TYPE "CLEANING HOPPER"
// stored: IsFailsafeCompliant false
   STRUCT
      FAULTED : Bool;
      "START GENERAL CONDITIONS" : Bool;
      "START GENERAL CONDITIONS HELP" : Bool;
      "START INITIAL CONDITIONS" : Bool;
      "START INITIAL CONDITIONS HELP" : Bool;
      "START MANUAL REQUEST" : Bool;
      "FEEDBACK ON" : Bool;
      "START SEMI REQUEST" : Bool;
      "START AUTO REQUEST" : Bool;
      "START GLOBAL REQUEST" : Bool;
      "START COMMAND" : Bool;
      "SYSTEM ON" : Bool;
      "STOP GENERAL CONDITIONS" : Bool;
      "STOP GENERAL CONDITIONS HELP" : Bool;
      "STOP INITIAL CONDITIONS" : Bool;
      "STOP INITIAL CONDITIONS HELP" : Bool;
      "STOP MANUAL REQUEST" : Bool;
      "STOP SEMI REQUEST" : Bool;
      "STOP AUTO REQUEST" : Bool;
      "STOP GLOBAL REQUEST" : Bool;
      "STOP COMMAND" : Bool;
      STOPPED : Bool;
      "FEEDBACK OFF" : Bool;
   END_STRUCT;
END_TYPE

TYPE "FEED HOPPER"
// stored: IsFailsafeCompliant false
   STRUCT
      FAULTED : Bool;   // Faulted
      "START GENERAL CONDITIONS" : Bool;   // Start General Conditions
      "START GENERAL CONDITIONS HELP" : Bool;   // Start General Conditions Help
      "START INITIAL CONDITIONS" : Bool;   // Start Initial Conditions
      "START INITIAL CONDITIONS HELP" : Bool;   // Start Initial Conditions Help
      "START MANUAL REQUEST" : Bool;   // Start Manual Request
      "FEEDBACK ON" : Bool;   // Feedback On
      "START AUTO REQUEST" : Bool;   // Start Auto Request
      "START GLOBAL REQUEST" : Bool;   // Start Global Request
      "START COMMAND" : Bool;   // Start Command
      "SYSTEM ON" : Bool;   // System On
      "STOP GENERAL CONDITIONS" : Bool;   // Stop General Conditions
      "STOP GENERAL CONDITIONS HELP" : Bool;   // Stop General Conditions Help
      "STOP INITIAL CONDITIONS" : Bool;   // Stop Initial Conditions
      "STOP INITIAL CONDITIONS HELP" : Bool;   // Stop Initial Conditions Help
      "STOP MANUAL REQUEST" : Bool;   // Stop Manual Request
      "STOP AUTO REQUEST" : Bool;   // Stop Auto Request
      "STOP GLOBAL REQUEST" : Bool;   // Stop Global Request
      "STOP COMMAND" : Bool;   // Stop Command
      STOPPED : Bool;   // Stopped
      "FEEDBACK OFF" : Bool;   // Feedback Off
   END_STRUCT;
END_TYPE

TYPE "GENERAL_DATA_SEQUENCES"
// stored: IsFailsafeCompliant false
   STRUCT
      START_GENERAL_CONDITIONS : Bool;   // Start general conditions
      START_GENERAL_CONDITIONS_HELP : Bool;   // Start general conditions help
      START_INITIAL_CONDITIONS : Bool;   // Start initial conditions
      START_INITIAL_CONDITIONS_HELP : Bool;   // Start initial conditions help
      START_MANUAL_REQUEST : Bool;   // Start manual request
      START_PROGRAM_REQUEST : Bool;   // Start semi request
      START_AUTO_REQUEST : Bool;   // Start auto request
      START_COMMAND : Bool;   // Start command
      STOP_GENERAL_CONDITIONS : Bool;   // Stop general conditions
      STOP_GENERAL_CONDITIONS_HELP : Bool;   // Stop general conditions help
      STOP_INITIAL_CONDITIONS : Bool;   // Stop initial conditions
      STOP_INITIAL_CONDITIONS_HELP : Bool;   // Stop initial conditions help
      STOP_MANUAL_CONDITIONS : Bool;   // Stop manual conditions
      STOP_MANUAL_REQUEST : Bool;   // Stop manual request
      STOP_PROGRAM_REQUEST : Bool;   // Stop semi request
      STOP_AUTO_REQUEST : Bool;   // Stop auto request
      STOP_COMMAND : Bool;   // Stop command
      SEQUENCE_RUNNING : Bool;   // Sequence running
      STEP_1 : Bool;   // Step 1
      STEP_2 : Bool;   // Step 2
      STEP_3 : Bool;   // Step 3
      STEP_4 : Bool;   // Step 4
      STEP_5 : Bool;   // Step 5
      STEP_6 : Bool;   // Step 6
      STEP_7 : Bool;   // Step 7
      STEP_8 : Bool;   // Step 8
      STEP_9 : Bool;   // Step 9
      STEP_10 : Bool;   // Step 10
      STEP_11 : Bool;   // Step 11
      STEP_12 : Bool;   // Step 12
      RESET_PLC_SEQUENCE : Bool;   // Reset PLC sequence
      SEQUENCE_DONE : Bool;   // Sequence done
      SEQUENCE_EXCEEDED_TIME : Bool;   // Sequence exceeded time
      WARNING : Bool;   // Warning
   END_STRUCT;
END_TYPE

TYPE "GENERAL_DATA_START_STOP"
// stored: IsFailsafeCompliant false
   STRUCT
      START_GENERAL_CONDITIONS : Bool;   // Start general conditions
      START_GENERAL_CONDITIONS_HELP : Bool;   // Start general conditions help
      START_INITIAL_CONDITIONS : Bool;   // Start initial conditions
      START_INITIAL_CONDITIONS_HELP : Bool;   // Start initial conditions help
      START_MANUAL_REQUEST : Bool;   // Start manual request
      START_PROGRAM_REQUEST : Bool;   // Start program request
      START_AUTO_REQUEST : Bool;   // Start auto request
      START_GLOBAL_REQUEST : Bool;   // Start global request
      START_COMMAND : Bool;   // Start command
      FEEDBACK_ON : Bool;   // Feedback on
      SYSTEM_ON : Bool;   // System on
      STOP_GENERAL_CONDITIONS : Bool;   // Stop general conditions
      STOP_GENERAL_CONDITIONS_HELP : Bool;   // Stop general conditions help
      STOP_INITIAL_CONDITIONS : Bool;   // Stop initial conditions
      STOP_INITIAL_CONDITIONS_HELP : Bool;   // Stop initial conditions help
      STOP_MANUAL_REQUEST : Bool;   // Stop manual request
      STOP_PROGRAM_REQUEST : Bool;   // Stop program request
      STOP_AUTO_REQUEST : Bool;   // Stop auto request
      STOP_GLOBAL_REQUEST : Bool;   // Stop global request
      STOP_COMMAND : Bool;   // Stop command
      FEEDBACK_OFF : Bool;   // Feedback off
      SYSTEM_OFF : Bool;   // System off
      FAULT : Bool;   // Fault
   END_STRUCT;
END_TYPE

TYPE "HMI_DATA_START_STOP"
// stored: IsFailsafeCompliant false
   STRUCT
      HMI_START : Bool;   // HMI start
      HMI_STOP : Bool;   // HMI stop
      HMI_STARTED : Bool;   // HMI started
      HMI_STOPPED : Bool;   // HMI stopped
      HMI_STARTING : Bool;   // HMI starting
      HMI_STOPPING : Bool;   // HMI stopping
      HMI_START_CONDITIONS : Bool;   // HMI start conditions
      HMI_STOP_CONDITIONS : Bool;   // HMI stop conditions
   END_STRUCT;
END_TYPE

TYPE "HOPPER PRESSURE CONTROL"
// stored: IsFailsafeCompliant false
   STRUCT
      FAULTED : Bool;
      "START GENERAL CONDITIONS" : Bool;
      "START GENERAL CONDITIONS HELP" : Bool;
      "START INITIAL CONDITIONS" : Bool;
      "START INITIAL CONDITIONS HELP" : Bool;
      "START MANUAL REQUEST" : Bool;
      "FEEDBACK ON" : Bool;
      "START AUTO REQUEST" : Bool;
      "START GLOBAL REQUEST" : Bool;
      "START COMMAND" : Bool;
      "SYSTEM ON" : Bool;
      "STOP GENERAL CONDITIONS" : Bool;
      "STOP GENERAL CONDITIONS HELP" : Bool;
      "STOP INITIAL CONDITIONS" : Bool;
      "STOP INITIAL CONDITIONS HELP" : Bool;
      "STOP MANUAL REQUEST" : Bool;
      "STOP AUTO REQUEST" : Bool;
      "STOP GLOBAL REQUEST" : Bool;
      "STOP COMMAND" : Bool;
      STOPPED : Bool;
      "FEEDBACK OFF" : Bool;
      "CONTROL DONE" : Bool;
      "SETPOINT PRESSURE" : Real;
      "FEEDBACK PRESSURE" : Real;
      "LIM LO" : Real;
      "LIM HI" : Real;
      "HMI START" : Bool;
      "HMI STOP" : Bool;
      "HMI START CONDITIONS" : Bool;
      "HMI STOP CONDITIONS" : Bool;
      "HMI STARTED" : Bool;
      "HMI STOPPED" : Bool;
      "HMI STARTING" : Bool;
      "HMI STOPPING" : Bool;
      "HMI PRESSURE VALUE" : Real;
      HMI_PRESSURE_INCREMENT : Real;
   END_STRUCT;
END_TYPE

TYPE "LOAD FEEDER SEQUENCE"
// stored: IsFailsafeCompliant false
   STRUCT
      "START GENERAL CONDITIONS" : Bool;   // General Conditions
      "START INITIAL CONDITIONS" : Bool;   // Initial Conditions
      "START SEMI REQUEST" : Bool;   // Semi Start Request
      "START AUTO REQUEST" : Bool;   // Auto Start Request
      "START COMMAND" : Bool;   // Global Start Request
      "STOP GENERAL CONDITIONS" : Bool;   // General Conditions
      "STOP INITIAL CONDITIONS" : Bool;   // Initial Conditions
      "STOP SEMI REQUEST" : Bool;   // Semi Start Request
      "STOP AUTO REQUEST" : Bool;   // Auto Start Request
      "STOP COMMAND" : Bool;   // Global Start Request
      "SEQUENCE RUNNING" : Bool;   // Sequence Running
      "STEP 1" : Bool;   // Step 1
      "STEP 2" : Bool;   // Step 2
      "STEP 3" : Bool;   // Step 3
      "STEP 4" : Bool;   // Step 4
      "STEP 5" : Bool;   // Step 5
      "STEP 6" : Bool;   // Step 6
      "STEP 7" : Bool;   // Step 7
      "RESET PLC SEQUENCE" : Bool;   // Reset PLC Sequence
      "REQUEST START VALVE" : Bool;   // Semi Auto Request
      "REQUEST STOP VALVE" : Bool;
      "REQUEST START PRESSURE" : Bool;   // Semi Auto Request
      "REQUESTE STOP PRESSURE" : Bool;
      "SETPOINT PRESSURE" : Real;
      "PASS STEP" : Bool;
      "SEQUENCE DONE" : Bool;   // Sequence Done
      WARNING : Bool;   // Warning
      "START GENERAL CONDITIONS HELP" : Bool;   // General Conditions Help
      "START INITIAL CONDITIONS HELP" : Bool;   // Initial Conditions Help
      "STOP GENERAL CONDITIONS HELP" : Bool;   // General Conditions Help
      "STOP INITIAL CONDITIONS HELP" : Bool;   // Initial Conditions Help
      "WARNING GONE" : Bool;   // Warning Gone
      "TIME ACTION" : Time;
      "APPLIED TIME ACTION" : Bool;
      "HMI START CONDITIONS" : Bool;   // HMI Start Conditions
      "HMI STOP CONDITIONS" : Bool;   // HMI Stop Conditions
      "HMI SEQUENCE RUNNING" : Bool;   // HMI Sequence Running
      "HMI SEQUENCE DONE" : Bool;   // HMI Sequence Done
      "HMI TIME LOAD" : UDInt;   // HMI Time Load
      "HMI FEEDBACK TIMER LOAD" : Int;
   END_STRUCT;
END_TYPE

TYPE "MOTOR_CONTROL_DATA"
// stored: IsFailsafeCompliant false
   STRUCT
      Start : Bool;
      Conditions : Bool;
      CCW_Rotation : Bool;
      CW_Rotation : Bool;
      "Manual Speed" : Real;
      "Consignment Speed" : Real;
      Min_Range : Real;
      Max_Range : Real;
      Lim_Lo : Real;
      Lim_HI : Real;
      Analog_Lo : Real;
      Analog_Hi : Real;
      "HMI Manual Cons." : Real;
      "HMI Consignment" : Real;
      "HMI Feedback Value" : Real;
   END_STRUCT;
END_TYPE

TYPE "HMI_ACTUATOR"
// stored: IsFailsafeCompliant false
   STRUCT
      HMI_START : Bool;
      HMI_STOP : Bool;
      HMI_START_CONDITIONS : Bool;
      HMI_STOP_CONDITIONS : Bool;
      HMI_STARTED : Bool;
      HMI_STOPPED : Bool;
      HMI_STARTING : Bool;
      HMI_STOPPING : Bool;
   END_STRUCT;
END_TYPE

TYPE "HMI_MACHINE_OVERVIEW"
// stored: IsFailsafeCompliant false
   STRUCT
      E_STOP_ROBOT : Bool;
      E_STOP_LASER : Bool;
      E_STOP_MAIN_PANEL : Bool;
      E_STOP_MAIN_SAFETY_DOOR : Bool;
      E_STOP_CELL : Bool;
      E_STOP_AUTOMATIC_DOOR : Bool;
      SAFETY_DOOR_L : Bool;
      SAFETY_DOOR_r : Bool;
      MAIN_SAFETY_DOOR : Bool;
      ANALOG_MODE_ON : Bool;
      CONTROL_SPARE_12 : Bool;
      CONTROL_SPARE_13 : Bool;
      CONTROL_SPARE_14 : Bool;
      CONTROL_SPARE_15 : Bool;
      CONTROL_SPARE_16 : Bool;
      CONTROL_SPARE_17 : Bool;
      COMMAND_POWER : DInt;
      REAL_POWER : DInt;
      PYROMETER_ACTUAL_TEMP : Real;
      LENS_HOLDER_FLOW : Real;
      LENS_HOLDER_TEMP : Real;
      ADITIVE_NOZZLE_FLOW : Real;
      ADITIVE_NOZZLE_TEMP : Real;
      DATA7 : DInt;
      DATA8 : DInt;
      DATA9 : Real;
      DATA10 : Real;
      DATA11 : Real;
      DATA12 : Real;
   END_STRUCT;
END_TYPE

TYPE "HMI_SERVICE"
// stored: IsFailsafeCompliant false
   STRUCT
      HMI_START : Bool;
      HMI_STOP : Bool;
      HMI_STARTING : Bool;
      HMI_STOPPING : Bool;
      HMI_STARTED : Bool;
      HMI_STOPPED : Bool;
      HMI_START_CONDITIONS : Bool;
      HMI_STOP_CONDITIONS : Bool;
      FAULTED : Bool;
   END_STRUCT;
END_TYPE

TYPE "AXIS"
// stored: IsFailsafeCompliant false
   STRUCT
      ENABLED : Bool;   // ENABLED
      SELECTED : Bool;   // SELECTED
      HMI_JOG_MINUS_RQ : Bool;   // HMI JOG MINUS RQ
      HMI_JOG_PLUS_RQ : Bool;   // HMI JOG PLUS RQ
      HMI_JOG_MINUS_CMM : Bool;   // HMI JOG MINUS COMMAND
      HMI_JOG_PLUS_CMM : Bool;   // HMI JOG PLUS COMMAND
      AUTO_RETURN_CMM : Bool;   // AUTO RETURN COMMAND
      AUTO_ADVANCE_CMM : Bool;   // AUTO ADVANCE COMMAND
      JOG_HELP : Bool;   // JOG HELP
      MINUS_BUTTON_HELP : Bool;   // MINUS BUTTON HELP
      PLUS_BUTTON_HELP : Bool;   // PLUS BUTTON HELP
      OPERATOR_HELP : Bool;   // OPERATOR HELP
      P1_TRIGGER : Bool;   // P1 TRIGGER
      P2_TRIGGER : Bool;   // P2 TRIGGER
      N1_TRIGGER : Bool;   // N1 TRIGGER
      N2_TRIGGER : Bool;   // N2 TRIGGER
      POS_TO_GO_FC18 : Real;   // POS TO GO FC18
      FC18_AXIS_IN_POS : Bool;   // FC18 AXIS IN POSITION
      FC18_FAULT : Bool;   // FC18 FAULT
      E_GANT_GROUP_SYN : Bool;   // GANTRY GROUP IS SYNCRONOUS
   END_STRUCT;
END_TYPE

TYPE "SPINDLE"
// stored: IsFailsafeCompliant false
   STRUCT
      SELECTED { ExternalVisible := 'False'; ExternalWritable := 'False'} : Bool;   // SELECTED
      CONT_INCRMTL_MODE { ExternalVisible := 'False'; ExternalWritable := 'False'} : Bool;   // CONTINOUS INCRMTL MODE
      HMI_JOG_MINUS_RQ { ExternalVisible := 'False'; ExternalWritable := 'False'} : Bool;   // HMI JOG MINUS REQUEST
      HMI_JOG_PLUS_RQ { ExternalVisible := 'False'; ExternalWritable := 'False'} : Bool;   // HMI JOG PLUS REQUEST
      HMI_JOG_MINUS_CMM { ExternalVisible := 'False'; ExternalWritable := 'False'} : Bool;   // HMI JOG MINUS COMMAND
      HMI_JOG_PLUS_CMM { ExternalVisible := 'False'; ExternalWritable := 'False'} : Bool;   // HMI JOG PLUS COMMAND
      SPEED_REACHED { ExternalVisible := 'False'; ExternalWritable := 'False'} : Bool;   // SPEED REACHED
      SPEED_ZERO { ExternalVisible := 'False'; ExternalWritable := 'False'} : Bool;   // SPEED ZERO
      JOG_HELP { ExternalVisible := 'False'; ExternalWritable := 'False'} : Bool;   // JOG HELP
      MINUS_BUTTON_HELP { ExternalVisible := 'False'; ExternalWritable := 'False'} : Bool;   // MINUS BUTTON HELP
      PLUS_BUTTON_HELP { ExternalVisible := 'False'; ExternalWritable := 'False'} : Bool;   // PLUS BUTTON HELP
      OPERATOR_HELP { ExternalVisible := 'False'; ExternalWritable := 'False'} : Bool;   // OPERATOR HELP
   END_STRUCT;
END_TYPE

TYPE "READ_DATA_MAG"
// stored: IsFailsafeCompliant false
   STRUCT
      FB2_DATA : Struct
         Error : Bool;   // Error
         Done : Bool;   // Done
         Request : Bool;   // Request
         Error_Fault : Bool;   // Error Fault
         Pulse : Bool;   // Pulse
         MAG_POS_IN_NC : Int;   // MAGAZINE POSITION IN NC
         Tool_state : Word;   // Tool state
         TOOL_NUMBER : Int;   // TOOL NUMBER
         MAGAZINE_POSITION : Int;   // MAGAZINE POSITION
      END_STRUCT;
      TOOL_DATA : Struct   // TOOL DATA
         NUM_CUTING_EDGE : Int;   // NUM CUTING EDGE
         QUANTITY_EDGE : Array[1..5] of Real;   // QUANTITY EDGE
         WARNING_EDGE : Array[1..5] of Real;   // WARNING EDGE
         EXPIRED_EDGE : Array[1..5] of Real;   // EXPIRED EDGE
      END_STRUCT;
      PARAM_MAGAZINE : Struct   // PARAM MAGAZINE
         TC_MOP4_QUANTITY_1 : Struct   // TC MOP4 QUANTITY 1
            SYNTAX_ID : Byte := BYTE#16#82;   // SYNTAX ID
            AREA_UNIT : Byte := BYTE#16#81;   // AREA UNIT
            COLUMN : Word := 16#0;   // TOOL NUMBER (HEX) / COLUMN
            LINE : Word := WORD#16#0004;   // $TC_MOP4[TOOL,1] CUTTING REMAINING LIFE COUNTER / LINE
            BLOCKTYPE : Byte := BYTE#16#22;   // BLOCKTYPE
            NUMOFLINE : Byte := BYTE#16#01;   // NUMOFLINE
            DATATYPE : Byte := BYTE#16#0F;   // DATATYPE
            LENGTH : Byte := BYTE#16#08;   // LENGTH
         END_STRUCT;
         TC_MOP4_QUANTITY_2 : Struct   // TC MOP4 QUANTITY 2
            SYNTAX_ID : Byte := BYTE#16#82;   // SYNTAX ID
            AREA_UNIT : Byte := BYTE#16#81;   // AREA UNIT
            COLUMN : Word := 16#0;   // TOOL NUMBER (HEX) / COLUMN
            LINE : Word := WORD#16#000D;   // $TC_MOP4[TOOL,2] CUTTING REMAINING LIFE COUNTER / LINE
            BLOCKTYPE : Byte := BYTE#16#22;   // BLOCKTYPE
            NUMOFLINE : Byte := BYTE#16#01;   // NUMOFLINE
            DATATYPE : Byte := BYTE#16#0F;   // DATATYPE
            LENGTH : Byte := BYTE#16#08;   // LENGTH
         END_STRUCT;
         TC_MOP4_QUANTITY_3 : Struct   // TC MOP4 QUANTITY 3
            SYNTAX_ID : Byte := BYTE#16#82;   // SYNTAX ID
            AREA_UNIT : Byte := BYTE#16#81;   // AREA UNIT
            COLUMN : Word := 16#0;   // TOOL NUMBER (HEX) / COLUMN
            LINE : Word := WORD#16#0016;   // $TC_MOP4[TOOL,3] CUTTING REMAINING LIFE COUNTER / LINE
            BLOCKTYPE : Byte := BYTE#16#22;   // BLOCKTYPE
            NUMOFLINE : Byte := BYTE#16#01;   // NUMOFLINE
            DATATYPE : Byte := BYTE#16#0F;   // DATATYPE
            LENGTH : Byte := BYTE#16#08;   // LENGTH
         END_STRUCT;
         TC_MOP4_QUANTITY_4 : Struct   // TC MOP4 QUANTITY 4
            SYNTAX_ID : Byte := BYTE#16#82;   // SYNTAX ID
            AREA_UNIT : Byte := BYTE#16#81;   // AREA UNIT
            COLUMN : Word := 16#0;   // TOOL NUMBER (HEX) / COLUMN
            LINE : Word := WORD#16#001F;   // $TC_MOP4[TOOL,4] CUTTING REMAINING LIFE COUNTER / LINE
            BLOCKTYPE : Byte := BYTE#16#22;   // BLOCKTYPE
            NUMOFLINE : Byte := BYTE#16#01;   // NUMOFLINE
            DATATYPE : Byte := BYTE#16#0F;   // DATATYPE
            LENGTH : Byte := BYTE#16#08;   // LENGTH
         END_STRUCT;
         TC_MOP4_QUANTITY_5 : Struct   // TC MOP4 QUANTITY 5
            SYNTAX_ID : Byte := BYTE#16#82;   // SYNTAX ID
            AREA_UNIT : Byte := BYTE#16#81;   // AREA UNIT
            COLUMN : Word := 16#0;   // TOOL NUMBER (HEX) / COLUMN
            LINE : Word := WORD#16#0028;   // $TC_MOP4[TOOL,4] CUTTING REMAINING LIFE COUNTER / LINE
            BLOCKTYPE : Byte := BYTE#16#22;   // BLOCKTYPE
            NUMOFLINE : Byte := BYTE#16#01;   // NUMOFLINE
            DATATYPE : Byte := BYTE#16#0F;   // DATATYPE
            LENGTH : Byte := BYTE#16#08;   // LENGTH
         END_STRUCT;
         TC_MOP3_WARNING_1 : Struct   // TC MOP3 WARNING 1
            SYNTAX_ID : Byte := BYTE#16#82;   // SYNTAX ID
            AREA_UNIT : Byte := BYTE#16#81;   // AREA UNIT
            COLUMN : Word := 16#0;   // TOOL NUMBER (HEX) / COLUMN
            LINE : Word := WORD#16#0003;   // $TC_MOP3[TOOL,1] CUTTING PREWARNING LIFE COUNTER / LINE
            BLOCKTYPE : Byte := BYTE#16#22;   // BLOCKTYPE
            NUMOFLINE : Byte := BYTE#16#01;   // NUMOFLINE
            DATATYPE : Byte := BYTE#16#0F;   // DATATYPE
            LENGTH : Byte := BYTE#16#08;   // LENGTH
         END_STRUCT;
         TC_MOP3_WARNING_2 : Struct   // TC MOP3 WARNING 2
            SYNTAX_ID : Byte := BYTE#16#82;   // SYNTAX ID
            AREA_UNIT : Byte := BYTE#16#81;   // AREA UNIT
            COLUMN : Word := 16#0;   // TOOL NUMBER (HEX) / COLUMN
            LINE : Word := WORD#16#000C;   // $TC_MOP3[TOOL,2] CUTTING PREWARNING LIFE COUNTER / LINE
            BLOCKTYPE : Byte := BYTE#16#22;   // BLOCKTYPE
            NUMOFLINE : Byte := BYTE#16#01;   // NUMOFLINE
            DATATYPE : Byte := BYTE#16#0F;   // DATATYPE
            LENGTH : Byte := BYTE#16#08;   // LENGTH
         END_STRUCT;
         TC_MOP3_WARNING_3 : Struct   // TC MOP3 WARNING 3
            SYNTAX_ID : Byte := BYTE#16#82;   // SYNTAX ID
            AREA_UNIT : Byte := BYTE#16#81;   // AREA UNIT
            COLUMN : Word := 16#0;   // TOOL NUMBER (HEX) / COLUMN
            LINE : Word := WORD#16#0015;   // $TC_MOP3[TOOL,3] CUTTING PREWARNING LIFE COUNTER / LINE
            BLOCKTYPE : Byte := BYTE#16#22;   // BLOCKTYPE
            NUMOFLINE : Byte := BYTE#16#01;   // NUMOFLINE
            DATATYPE : Byte := BYTE#16#0F;   // DATATYPE
            LENGTH : Byte := BYTE#16#08;   // LENGTH
         END_STRUCT;
         TC_MOP3_WARNING_4 : Struct   // TC MOP3 WARNING 4
            SYNTAX_ID : Byte := BYTE#16#82;   // SYNTAX ID
            AREA_UNIT : Byte := BYTE#16#81;   // AREA UNIT
            COLUMN : Word := 16#0;   // TOOL NUMBER (HEX) / COLUMN
            LINE : Word := WORD#16#001E;   // $TC_MOP3[TOOL,4] CUTTING PREWARNING LIFE COUNTER / LINE
            BLOCKTYPE : Byte := BYTE#16#22;   // BLOCKTYPE
            NUMOFLINE : Byte := BYTE#16#01;   // NUMOFLINE
            DATATYPE : Byte := BYTE#16#0F;   // DATATYPE
            LENGTH : Byte := BYTE#16#08;   // LENGTH
         END_STRUCT;
         TC_MOP3_WARNING_5 : Struct   // TC MOP3 WARNING 5
            SYNTAX_ID : Byte := BYTE#16#82;   // SYNTAX ID
            AREA_UNIT : Byte := BYTE#16#81;   // AREA UNIT
            COLUMN : Word := 16#0;   // TOOL NUMBER (HEX) / COLUMN
            LINE : Word := WORD#16#0027;   // $TC_MOP3[TOOL,4] CUTTING PREWARNING LIFE COUNTER / LINE
            BLOCKTYPE : Byte := BYTE#16#22;   // BLOCKTYPE
            NUMOFLINE : Byte := BYTE#16#01;   // NUMOFLINE
            DATATYPE : Byte := BYTE#16#0F;   // DATATYPE
            LENGTH : Byte := BYTE#16#08;   // LENGTH
         END_STRUCT;
         TC_MOP13_EXPIRED_1 : Struct   // TC MOP13 EXPIRED 1
            SYNTAX_ID : Byte := BYTE#16#82;   // SYNTAX ID
            AREA_UNIT : Byte := BYTE#16#81;   // AREA UNIT
            COLUMN : Word := 16#0;   // TOOL NUMBER (HEX) / COLUMN
            LINE : Word := WORD#16#0006;   // $TC_MOP13[TOOL,1] CUTTING SET POINT LIFE COUNTER / LINE
            BLOCKTYPE : Byte := BYTE#16#22;   // BLOCKTYPE
            NUMOFLINE : Byte := BYTE#16#01;   // NUMOFLINE
            DATATYPE : Byte := BYTE#16#0F;   // DATATYPE
            LENGTH : Byte := BYTE#16#08;   // LENGTH
         END_STRUCT;
         TC_MOP13_EXPIRED_2 : Struct   // TC MOP13 EXPIRED 2
            SYNTAX_ID : Byte := BYTE#16#82;   // SYNTAX ID
            AREA_UNIT : Byte := BYTE#16#81;   // AREA UNIT
            COLUMN : Word := 16#0;   // TOOL NUMBER (HEX) / COLUMN
            LINE : Word := WORD#16#000F;   // $TC_MOP13[TOOL,2] CUTTING SET POINT LIFE COUNTER / LINE
            BLOCKTYPE : Byte := BYTE#16#22;   // BLOCKTYPE
            NUMOFLINE : Byte := BYTE#16#01;   // NUMOFLINE
            DATATYPE : Byte := BYTE#16#0F;   // DATATYPE
            LENGTH : Byte := BYTE#16#08;   // LENGTH
         END_STRUCT;
         TC_MOP13_EXPIRED_3 : Struct   // TC MOP13 EXPIRED 3
            SYNTAX_ID : Byte := BYTE#16#82;   // SYNTAX ID
            AREA_UNIT : Byte := BYTE#16#81;   // AREA UNIT
            COLUMN : Word := 16#0;   // TOOL NUMBER (HEX) / COLUMN
            LINE : Word := WORD#16#0018;   // $TC_MOP13[TOOL,3] CUTTING SET POINT LIFE COUNTER / LINE
            BLOCKTYPE : Byte := BYTE#16#22;   // BLOCKTYPE
            NUMOFLINE : Byte := BYTE#16#01;   // NUMOFLINE
            DATATYPE : Byte := BYTE#16#0F;   // DATATYPE
            LENGTH : Byte := BYTE#16#08;   // LENGTH
         END_STRUCT;
         TC_MOP13_EXPIRED_4 : Struct   // TC MOP13 EXPIRED 4
            SYNTAX_ID : Byte := BYTE#16#82;   // SYNTAX ID
            AREA_UNIT : Byte := BYTE#16#81;   // AREA UNIT
            COLUMN : Word := 16#0;   // TOOL NUMBER (HEX) / COLUMN
            LINE : Word := WORD#16#0021;   // $TC_MOP13[TOOL,4] CUTTING SET POINT LIFE COUNTER / LINE
            BLOCKTYPE : Byte := BYTE#16#22;   // BLOCKTYPE
            NUMOFLINE : Byte := BYTE#16#01;   // NUMOFLINE
            DATATYPE : Byte := BYTE#16#0F;   // DATATYPE
            LENGTH : Byte := BYTE#16#08;   // LENGTH
         END_STRUCT;
         TC_MOP13_EXPIRED_5 : Struct   // TC MOP13 EXPIRED 5
            SYNTAX_ID : Byte := BYTE#16#82;   // SYNTAX ID
            AREA_UNIT : Byte := BYTE#16#81;   // AREA UNIT
            COLUMN : Word := 16#0;   // TOOL NUMBER (HEX) / COLUMN
            LINE : Word := WORD#16#002A;   // $TC_MOP13[TOOL,4] CUTTING SET POINT LIFE COUNTER / LINE
            BLOCKTYPE : Byte := BYTE#16#22;   // BLOCKTYPE
            NUMOFLINE : Byte := BYTE#16#01;   // NUMOFLINE
            DATATYPE : Byte := BYTE#16#0F;   // DATATYPE
            LENGTH : Byte := BYTE#16#08;   // LENGTH
         END_STRUCT;
      END_STRUCT;
      FB2_VARS : Struct   // FB2 VARS
         TOOL_NUMBER : Struct   // TOOL NUMBER
            error : Bool;   // error
            done : Bool;   // done
            request : Bool;   // request
         END_STRUCT;
         ORIGI_MAGAZINE : Struct   // ORIGI MAGAZINE
            error : Bool;   // error
            done : Bool;   // done
            request : Bool;   // request
         END_STRUCT;
         CUTING_EDGE : Struct   // CUTING EDGE
            error : Bool;   // error
            done : Bool;   // done
            request : Bool;   // request
         END_STRUCT;
         QUANTITY_EDGE : Struct   // QUANTITY EDGE
            error : Bool;   // error
            done : Bool;   // done
            request : Bool;   // request
         END_STRUCT;
         WARNING_EDGE : Struct   // WARNING EDGE
            error : Bool;   // error
            done : Bool;   // done
            request : Bool;   // request
         END_STRUCT;
         EXPIRED_EDGE : Struct   // EXPIRED EDGE
            error : Bool;   // error
            done : Bool;   // done
            request : Bool;   // request
         END_STRUCT;
      END_STRUCT;
      SMNS_PRMTS_MAG : Struct   // SMNS PRMTS MAG
         MAG_DATA_TC_MPP6_PLACE_DATA : Struct   // MAG DATA TC MPP6 PLACE DATA
            SYNTAX_ID : Byte := BYTE#16#82;   // SYNTAX ID
            AREA_UNIT : Byte := BYTE#16#81;   // CHANNEL NUMBER, 81=CH1, 82=CH2 ) / AREA UNIT
            COLUMN : Word := WORD#16#0001;   // MAGAZINE NUMBER / COLUMN
            LINE : Word := 16#0;   // LINE
            BLOCKTYPE : Byte := BYTE#16#28;   // BLOCKTYPE
            NUMOFLINE : Byte := BYTE#16#01;   // NUMOFLINE
            DATATYPE : Byte := BYTE#16#04;   // DATATYPE
            LENGTH : Byte := BYTE#16#02;   // LENGTH
         END_STRUCT;
         MAG_DATA_NUM_CUTTING_EDGES : Struct   // MAG DATA NUM CUTTING EDGES
            SYNTAX_ID : Byte := BYTE#16#82;   // SYNTAX ID
            AREA_UNIT : Byte := BYTE#16#81;   // AREA UNIT
            COLUMN : Word := WORD#16#000E;   // NUM CUTTING EDGES / COLUMN
            LINE : Word := WORD#16#0001;   // LINE
            BLOCKTYPE : Byte := BYTE#16#21;   // BLOCKTYPE
            NUMOFLINE : Byte := BYTE#16#01;   // NUMOFLINE
            DATATYPE : Byte := BYTE#16#04;   // DATATYPE
            LENGTH : Byte := BYTE#16#02;   // LENGTH
         END_STRUCT;
      END_STRUCT;
   END_STRUCT;
   // // TOOL_DATA.QUANTITY_EDGE[1] : QUANTITY EDGE[1]
   // // TOOL_DATA.QUANTITY_EDGE[2] : QUANTITY EDGE[2]
   // // TOOL_DATA.QUANTITY_EDGE[3] : QUANTITY EDGE[3]
   // // TOOL_DATA.QUANTITY_EDGE[4] : QUANTITY EDGE[4]
   // // TOOL_DATA.QUANTITY_EDGE[5] : QUANTITY EDGE[5]
   // // TOOL_DATA.WARNING_EDGE[1] : WARNING EDGE[1]
   // // TOOL_DATA.WARNING_EDGE[2] : WARNING EDGE[2]
   // // TOOL_DATA.WARNING_EDGE[3] : WARNING EDGE[3]
   // // TOOL_DATA.WARNING_EDGE[4] : WARNING EDGE[4]
   // // TOOL_DATA.WARNING_EDGE[5] : WARNING EDGE[5]
   // // TOOL_DATA.EXPIRED_EDGE[1] : EXPIRED EDGE[1]
   // // TOOL_DATA.EXPIRED_EDGE[2] : EXPIRED EDGE[2]
   // // TOOL_DATA.EXPIRED_EDGE[3] : EXPIRED EDGE[3]
   // // TOOL_DATA.EXPIRED_EDGE[4] : EXPIRED EDGE[4]
   // // TOOL_DATA.EXPIRED_EDGE[5] : EXPIRED EDGE[5]
END_TYPE

TYPE "READ_TOOL_DATA_SP1"
// stored: IsFailsafeCompliant false
   STRUCT
      READ : Struct
         FB2_DATA_SP1 : Struct
            Error : Bool;   // Error
            Done : Bool;   // Done
            Request : Bool;   // Request
            Error_Fault : Bool;   // Error Fault
            Status : Word;   // Pulse
            MAG_POS_IN_NC : Int;   // MAGAZINE POSITION IN NC
            Tool_state : Word;   // Tool state
            TOOL_NUMBER : Int;   // TOOL NUMBER
            MAGAZINE_POSITION : Int;   // MAGAZINE POSITION
         END_STRUCT;
         TOOL_DATA_SP1 : Struct   // TOOL DATA
            NUM_CUTING_EDGE : Int;   // NUM CUTING EDGE
            QUANTITY_EDGE : Array[1..5] of Real;   // QUANTITY EDGE
            WARNING_EDGE : Array[1..5] of Real;   // WARNING EDGE
            EXPIRED_EDGE : Array[1..5] of Real;   // EXPIRED EDGE
         END_STRUCT;
         PARAM_SPINDLE_SP1 : Struct
            TC_MOP4_QUANTITY_1 : Struct
               SYNTAX_ID : Byte := BYTE#16#82;   // SYNTAX ID
               AREA_UNIT : Byte := BYTE#16#81;   // AREA UNIT
               COLUMN : Word := 16#0;   // TOOL NUMBER (HEX)
               LINE : Word := WORD#16#0004;   // $TC_MOP4[TOOL,1] CUTTING REMAINING LIFE COUNTER
               BLOCKTYPE : Byte := BYTE#16#22;   // BLOCKTYPE
               NUMOFLINE : Byte := BYTE#16#01;   // NUMOFLINE
               DATATYPE : Byte := BYTE#16#0F;   // DATATYPE
               LENGTH : Byte := BYTE#16#08;   // LENGTH
            END_STRUCT;
            TC_MOP4_QUANTITY_2 : Struct
               SYNTAX_ID : Byte := BYTE#16#82;
               AREA_UNIT : Byte := BYTE#16#81;
               COLUMN : Word := 16#0;   // TOOL NUMBER (HEX)
               LINE : Word := WORD#16#000D;   // $TC_MOP4[TOOL,2] CUTTING REMAINING LIFE COUNTER
               BLOCKTYPE : Byte := BYTE#16#22;
               NUMOFLINE : Byte := BYTE#16#01;
               DATATYPE : Byte := BYTE#16#0F;
               LENGTH : Byte := BYTE#16#08;
            END_STRUCT;
            TC_MOP4_QUANTITY_3 : Struct
               SYNTAX_ID : Byte := BYTE#16#82;
               AREA_UNIT : Byte := BYTE#16#81;
               COLUMN : Word := 16#0;   // TOOL NUMBER (HEX)
               LINE : Word := WORD#16#0016;   // $TC_MOP4[TOOL,3] CUTTING REMAINING LIFE COUNTER
               BLOCKTYPE : Byte := BYTE#16#22;
               NUMOFLINE : Byte := BYTE#16#01;
               DATATYPE : Byte := BYTE#16#0F;
               LENGTH : Byte := BYTE#16#08;
            END_STRUCT;
            TC_MOP4_QUANTITY_4 : Struct
               SYNTAX_ID : Byte := BYTE#16#82;
               AREA_UNIT : Byte := BYTE#16#81;
               COLUMN : Word := 16#0;   // TOOL NUMBER (HEX)
               LINE : Word := WORD#16#001F;   // $TC_MOP4[TOOL,4] CUTTING REMAINING LIFE COUNTER
               BLOCKTYPE : Byte := BYTE#16#22;
               NUMOFLINE : Byte := BYTE#16#01;
               DATATYPE : Byte := BYTE#16#0F;
               LENGTH : Byte := BYTE#16#08;
            END_STRUCT;
            TC_MOP4_QUANTITY_5 : Struct
               SYNTAX_ID : Byte := BYTE#16#82;
               AREA_UNIT : Byte := BYTE#16#81;
               COLUMN : Word := 16#0;   // TOOL NUMBER (HEX)
               LINE : Word := WORD#16#0028;   // $TC_MOP4[TOOL,4] CUTTING REMAINING LIFE COUNTER / $TC_MOP4[TOOL,5] CUTTING REMAINING LIFE COUNTER
               BLOCKTYPE : Byte := BYTE#16#22;
               NUMOFLINE : Byte := BYTE#16#01;
               DATATYPE : Byte := BYTE#16#0F;
               LENGTH : Byte := BYTE#16#08;
            END_STRUCT;
            TC_MOP3_WARNING_1 : Struct
               SYNTAX_ID : Byte := BYTE#16#82;
               AREA_UNIT : Byte := BYTE#16#81;
               COLUMN : Word := 16#0;   // TOOL NUMBER (HEX)
               LINE : Word := WORD#16#0003;   // $TC_MOP3[TOOL,1] CUTTING PREWARNING LIFE COUNTER
               BLOCKTYPE : Byte := BYTE#16#22;
               NUMOFLINE : Byte := BYTE#16#01;
               DATATYPE : Byte := BYTE#16#0F;
               LENGTH : Byte := BYTE#16#08;
            END_STRUCT;
            TC_MOP3_WARNING_2 : Struct
               SYNTAX_ID : Byte := BYTE#16#82;
               AREA_UNIT : Byte := BYTE#16#81;
               COLUMN : Word := 16#0;   // TOOL NUMBER (HEX)
               LINE : Word := WORD#16#000C;   // $TC_MOP3[TOOL,2] CUTTING PREWARNING LIFE COUNTER
               BLOCKTYPE : Byte := BYTE#16#22;
               NUMOFLINE : Byte := BYTE#16#01;
               DATATYPE : Byte := BYTE#16#0F;
               LENGTH : Byte := BYTE#16#08;
            END_STRUCT;
            TC_MOP3_WARNING_3 : Struct
               SYNTAX_ID : Byte := BYTE#16#82;
               AREA_UNIT : Byte := BYTE#16#81;
               COLUMN : Word := 16#0;   // TOOL NUMBER (HEX)
               LINE : Word := WORD#16#0015;   // $TC_MOP3[TOOL,3] CUTTING PREWARNING LIFE COUNTER
               BLOCKTYPE : Byte := BYTE#16#22;
               NUMOFLINE : Byte := BYTE#16#01;
               DATATYPE : Byte := BYTE#16#0F;
               LENGTH : Byte := BYTE#16#08;
            END_STRUCT;
            TC_MOP3_WARNING_4 : Struct
               SYNTAX_ID : Byte := BYTE#16#82;
               AREA_UNIT : Byte := BYTE#16#81;
               COLUMN : Word := 16#0;   // TOOL NUMBER (HEX)
               LINE : Word := WORD#16#001E;   // $TC_MOP3[TOOL,4] CUTTING PREWARNING LIFE COUNTER
               BLOCKTYPE : Byte := BYTE#16#22;
               NUMOFLINE : Byte := BYTE#16#01;
               DATATYPE : Byte := BYTE#16#0F;
               LENGTH : Byte := BYTE#16#08;
            END_STRUCT;
            TC_MOP3_WARNING_5 : Struct
               SYNTAX_ID : Byte := BYTE#16#82;
               AREA_UNIT : Byte := BYTE#16#81;
               COLUMN : Word := 16#0;   // TOOL NUMBER (HEX)
               LINE : Word := WORD#16#0027;   // $TC_MOP3[TOOL,4] CUTTING PREWARNING LIFE COUNTER / $TC_MOP3[TOOL,5] CUTTING PREWARNING LIFE COUNTER
               BLOCKTYPE : Byte := BYTE#16#22;
               NUMOFLINE : Byte := BYTE#16#01;
               DATATYPE : Byte := BYTE#16#0F;
               LENGTH : Byte := BYTE#16#08;
            END_STRUCT;
            TC_MOP13_EXPIRED_1 : Struct
               SYNTAX_ID : Byte := BYTE#16#82;
               AREA_UNIT : Byte := BYTE#16#81;
               COLUMN : Word := 16#0;   // TOOL NUMBER (HEX)
               LINE : Word := WORD#16#0006;   // $TC_MOP13[TOOL,1] CUTTING SET POINT LIFE COUNTER
               BLOCKTYPE : Byte := BYTE#16#22;
               NUMOFLINE : Byte := BYTE#16#01;
               DATATYPE : Byte := BYTE#16#0F;
               LENGTH : Byte := BYTE#16#08;
            END_STRUCT;
            TC_MOP13_EXPIRED_2 : Struct
               SYNTAX_ID : Byte := BYTE#16#82;
               AREA_UNIT : Byte := BYTE#16#81;
               COLUMN : Word := 16#0;   // TOOL NUMBER (HEX)
               LINE : Word := WORD#16#000F;   // $TC_MOP13[TOOL,2] CUTTING SET POINT LIFE COUNTER
               BLOCKTYPE : Byte := BYTE#16#22;
               NUMOFLINE : Byte := BYTE#16#01;
               DATATYPE : Byte := BYTE#16#0F;
               LENGTH : Byte := BYTE#16#08;
            END_STRUCT;
            TC_MOP13_EXPIRED_3 : Struct
               SYNTAX_ID : Byte := BYTE#16#82;
               AREA_UNIT : Byte := BYTE#16#81;
               COLUMN : Word := 16#0;   // TOOL NUMBER (HEX)
               LINE : Word := WORD#16#0018;   // $TC_MOP13[TOOL,3] CUTTING SET POINT LIFE COUNTER
               BLOCKTYPE : Byte := BYTE#16#22;
               NUMOFLINE : Byte := BYTE#16#01;
               DATATYPE : Byte := BYTE#16#0F;
               LENGTH : Byte := BYTE#16#08;
            END_STRUCT;
            TC_MOP13_EXPIRED_4 : Struct
               SYNTAX_ID : Byte := BYTE#16#82;
               AREA_UNIT : Byte := BYTE#16#81;
               COLUMN : Word := 16#0;   // TOOL NUMBER (HEX)
               LINE : Word := WORD#16#0021;   // $TC_MOP13[TOOL,4] CUTTING SET POINT LIFE COUNTER
               BLOCKTYPE : Byte := BYTE#16#22;
               NUMOFLINE : Byte := BYTE#16#01;
               DATATYPE : Byte := BYTE#16#0F;
               LENGTH : Byte := BYTE#16#08;
            END_STRUCT;
            TC_MOP13_EXPIRED_5 : Struct
               SYNTAX_ID : Byte := BYTE#16#82;
               AREA_UNIT : Byte := BYTE#16#81;
               COLUMN : Word := 16#0;   // TOOL NUMBER (HEX)
               LINE : Word := WORD#16#002A;   // $TC_MOP13[TOOL,4] CUTTING SET POINT LIFE COUNTER / $TC_MOP13[TOOL,5] CUTTING SET POINT LIFE COUNTER
               BLOCKTYPE : Byte := BYTE#16#22;
               NUMOFLINE : Byte := BYTE#16#01;
               DATATYPE : Byte := BYTE#16#0F;
               LENGTH : Byte := BYTE#16#08;
            END_STRUCT;
         END_STRUCT;
         FB2_VARS_SP1 : Struct
            TOOL_NUMBER : Struct
               error : Bool;
               done : Bool;
               request : Bool;
            END_STRUCT;
            ORIGI_MAGAZINE : Struct
               error : Bool;
               done : Bool;
               request : Bool;
            END_STRUCT;
            CUTING_EDGE : Struct
               error : Bool;
               done : Bool;
               request : Bool;
            END_STRUCT;
            QUANTITY_EDGE : Struct
               error : Bool;
               done : Bool;
               request : Bool;
            END_STRUCT;
            WARNING_EDGE : Struct
               error : Bool;
               done : Bool;
               request : Bool;
            END_STRUCT;
            EXPIRED_EDGE : Struct
               error : Bool;
               done : Bool;
               request : Bool;
            END_STRUCT;
         END_STRUCT;
         SMNS_PRMTRS_SP1 : Struct
            TC_MPP6_PLACE_DATA : Struct
               SYNTAX_ID : Byte := BYTE#16#82;
               AREA_UNIT : Byte := BYTE#16#81;   // CHANNEL NUMBER, 81=CH1, 82=CH2 )
               COLUMN : Word := WORD#16#0001;   // MAGAZINE NUMBER
               LINE : Word := 16#0;
               BLOCKTYPE : Byte := BYTE#16#28;
               NUMOFLINE : Byte := BYTE#16#01;
               DATATYPE : Byte := BYTE#16#04;
               LENGTH : Byte := BYTE#16#02;
            END_STRUCT;
            NUM_CUTTING_EDGES : Struct
               SYNTAX_ID : Byte := BYTE#16#82;
               AREA_UNIT : Byte := BYTE#16#81;
               COLUMN : Word := WORD#16#000E;   // NUM CUTTING EDGES
               LINE : Word := WORD#16#0001;
               BLOCKTYPE : Byte := BYTE#16#21;
               NUMOFLINE : Byte := BYTE#16#01;
               DATATYPE : Byte := BYTE#16#04;
               LENGTH : Byte := BYTE#16#02;
            END_STRUCT;
            DUPLO_NUMBER : Struct
               SYNTAX_ID : Byte := BYTE#16#82;
               AREA_UNIT : Byte := BYTE#16#81;
               COLUMN : Word := WORD#16#0002;   // DUPLO NUMBER
               LINE : Word := WORD#16#0001;
               BLOCKTYPE : Byte := BYTE#16#21;
               NUMOFLINE : Byte := BYTE#16#01;
               DATATYPE : Byte := BYTE#16#04;
               LENGTH : Byte := BYTE#16#02;
            END_STRUCT;
            ORIG_MAGAZINE : Struct
               SYNTAX_ID : Byte := BYTE#16#82;
               AREA_UNIT : Byte := BYTE#16#81;
               COLUMN : Word := WORD#16#0011;   // ORIG MAGAZINE
               LINE : Word := WORD#16#0001;
               BLOCKTYPE : Byte := BYTE#16#21;
               NUMOFLINE : Byte := BYTE#16#01;
               DATATYPE : Byte := BYTE#16#04;
               LENGTH : Byte := BYTE#16#02;
            END_STRUCT;
         END_STRUCT;
      END_STRUCT;
   END_STRUCT;
   // // READ.TOOL_DATA_SP1.QUANTITY_EDGE[1] : QUANTITY EDGE[1]
   // // READ.TOOL_DATA_SP1.QUANTITY_EDGE[2] : QUANTITY EDGE[2]
   // // READ.TOOL_DATA_SP1.QUANTITY_EDGE[3] : QUANTITY EDGE[3]
   // // READ.TOOL_DATA_SP1.QUANTITY_EDGE[4] : QUANTITY EDGE[4]
   // // READ.TOOL_DATA_SP1.QUANTITY_EDGE[5] : QUANTITY EDGE[5]
   // // READ.TOOL_DATA_SP1.WARNING_EDGE[1] : WARNING EDGE[1]
   // // READ.TOOL_DATA_SP1.WARNING_EDGE[2] : WARNING EDGE[2]
   // // READ.TOOL_DATA_SP1.WARNING_EDGE[3] : WARNING EDGE[3]
   // // READ.TOOL_DATA_SP1.WARNING_EDGE[4] : WARNING EDGE[4]
   // // READ.TOOL_DATA_SP1.WARNING_EDGE[5] : WARNING EDGE[5]
   // // READ.TOOL_DATA_SP1.EXPIRED_EDGE[1] : EXPIRED EDGE[1]
   // // READ.TOOL_DATA_SP1.EXPIRED_EDGE[2] : EXPIRED EDGE[2]
   // // READ.TOOL_DATA_SP1.EXPIRED_EDGE[3] : EXPIRED EDGE[3]
   // // READ.TOOL_DATA_SP1.EXPIRED_EDGE[4] : EXPIRED EDGE[4]
   // // READ.TOOL_DATA_SP1.EXPIRED_EDGE[5] : EXPIRED EDGE[5]
END_TYPE

TYPE "READ_TOOL_DATA_SP1_SP2"
// stored: IsFailsafeCompliant false
   STRUCT
      READ : Struct
         FB2_DATA_SP1 : Struct
            Error : Bool;   // Error
            Done : Bool;   // Done
            Request : Bool;   // Request
            Error_Fault : Bool;   // Error Fault
            Status : Word;   // Pulse
            MAG_POS_IN_NC : Int;   // MAGAZINE POSITION IN NC
            Tool_state : Word;   // Tool state
            TOOL_NUMBER : Int;   // TOOL NUMBER
            MAGAZINE_POSITION : Int;   // MAGAZINE POSITION
         END_STRUCT;
         FB2_DATA_SP2 : Struct
            Error : Bool;   // Error
            Done : Bool;   // Done
            Request : Bool;   // Request
            Error_Fault : Bool;   // Error Fault
            Status : Word;   // Pulse
            MAG_POS_IN_NC : Int;   // MAGAZINE POSITION IN NC
            Tool_state : Word;   // Tool state
            TOOL_NUMBER : Int;   // TOOL NUMBER
            MAGAZINE_POSITION : Int;   // MAGAZINE POSITION
         END_STRUCT;
         TOOL_DATA_SP1 : Struct
            NUM_CUTING_EDGE : Int;   // NUM CUTING EDGE
            QUANTITY_EDGE : Array[1..5] of Real;   // QUANTITY EDGE
            WARNING_EDGE : Array[1..5] of Real;   // WARNING EDGE
            EXPIRED_EDGE : Array[1..5] of Real;   // EXPIRED EDGE
         END_STRUCT;
         TOOL_DATA_SP2 : Struct
            NUM_CUTING_EDGE : Int;   // NUM CUTING EDGE
            QUANTITY_EDGE { ExternalAccessible := 'False'; ExternalVisible := 'False'; ExternalWritable := 'False'} : Array[1..5] of Real;   // QUANTITY EDGE
            WARNING_EDGE : Array[1..5] of Real;   // WARNING EDGE
            EXPIRED_EDGE : Array[1..5] of Real;   // EXPIRED EDGE
         END_STRUCT;
         PARAM_SPINDLE_SP1 : Struct
            TC_MOP4_QUANTITY_1 : Struct
               SYNTAX_ID : Byte := BYTE#16#82;
               AREA_UNIT : Byte := BYTE#16#81;
               COLUMN : Word := 16#0;   // TOOL NUMBER (HEX)
               LINE : Word := WORD#16#0004;   // $TC_MOP4[TOOL,1] CUTTING REMAINING LIFE COUNTER
               BLOCKTYPE : Byte := BYTE#16#22;
               NUMOFLINE : Byte := BYTE#16#01;
               DATATYPE : Byte := BYTE#16#0F;
               LENGTH : Byte := BYTE#16#08;
            END_STRUCT;
            TC_MOP4_QUANTITY_2 : Struct
               SYNTAX_ID : Byte := BYTE#16#82;
               AREA_UNIT : Byte := BYTE#16#81;
               COLUMN : Word := 16#0;   // TOOL NUMBER (HEX)
               LINE : Word := WORD#16#000D;   // $TC_MOP4[TOOL,2] CUTTING REMAINING LIFE COUNTER
               BLOCKTYPE : Byte := BYTE#16#22;
               NUMOFLINE : Byte := BYTE#16#01;
               DATATYPE : Byte := BYTE#16#0F;
               LENGTH : Byte := BYTE#16#08;
            END_STRUCT;
            TC_MOP4_QUANTITY_3 : Struct
               SYNTAX_ID : Byte := BYTE#16#82;
               AREA_UNIT : Byte := BYTE#16#81;
               COLUMN : Word := 16#0;   // TOOL NUMBER (HEX)
               LINE : Word := WORD#16#0016;   // $TC_MOP4[TOOL,3] CUTTING REMAINING LIFE COUNTER
               BLOCKTYPE : Byte := BYTE#16#22;
               NUMOFLINE : Byte := BYTE#16#01;
               DATATYPE : Byte := BYTE#16#0F;
               LENGTH : Byte := BYTE#16#08;
            END_STRUCT;
            TC_MOP4_QUANTITY_4 : Struct
               SYNTAX_ID : Byte := BYTE#16#82;
               AREA_UNIT : Byte := BYTE#16#81;
               COLUMN : Word := 16#0;   // TOOL NUMBER (HEX)
               LINE : Word := WORD#16#001F;   // $TC_MOP4[TOOL,4] CUTTING REMAINING LIFE COUNTER
               BLOCKTYPE : Byte := BYTE#16#22;
               NUMOFLINE : Byte := BYTE#16#01;
               DATATYPE : Byte := BYTE#16#0F;
               LENGTH : Byte := BYTE#16#08;
            END_STRUCT;
            TC_MOP4_QUANTITY_5 : Struct
               SYNTAX_ID : Byte := BYTE#16#82;
               AREA_UNIT : Byte := BYTE#16#81;
               COLUMN : Word := 16#0;   // TOOL NUMBER (HEX)
               LINE : Word := WORD#16#0028;   // $TC_MOP4[TOOL,4] CUTTING REMAINING LIFE COUNTER / $TC_MOP4[TOOL,5] CUTTING REMAINING LIFE COUNTER
               BLOCKTYPE : Byte := BYTE#16#22;
               NUMOFLINE : Byte := BYTE#16#01;
               DATATYPE : Byte := BYTE#16#0F;
               LENGTH : Byte := BYTE#16#08;
            END_STRUCT;
            TC_MOP3_WARNING_1 : Struct
               SYNTAX_ID : Byte := BYTE#16#82;
               AREA_UNIT : Byte := BYTE#16#81;
               COLUMN : Word := 16#0;   // TOOL NUMBER (HEX)
               LINE : Word := WORD#16#0003;   // $TC_MOP3[TOOL,1] CUTTING PREWARNING LIFE COUNTER
               BLOCKTYPE : Byte := BYTE#16#22;
               NUMOFLINE : Byte := BYTE#16#01;
               DATATYPE : Byte := BYTE#16#0F;
               LENGTH : Byte := BYTE#16#08;
            END_STRUCT;
            TC_MOP3_WARNING_2 : Struct
               SYNTAX_ID : Byte := BYTE#16#82;
               AREA_UNIT : Byte := BYTE#16#81;
               COLUMN : Word := 16#0;   // TOOL NUMBER (HEX)
               LINE : Word := WORD#16#000C;   // $TC_MOP3[TOOL,2] CUTTING PREWARNING LIFE COUNTER
               BLOCKTYPE : Byte := BYTE#16#22;
               NUMOFLINE : Byte := BYTE#16#01;
               DATATYPE : Byte := BYTE#16#0F;
               LENGTH : Byte := BYTE#16#08;
            END_STRUCT;
            TC_MOP3_WARNING_3 : Struct
               SYNTAX_ID : Byte := BYTE#16#82;
               AREA_UNIT : Byte := BYTE#16#81;
               COLUMN : Word := 16#0;   // TOOL NUMBER (HEX)
               LINE : Word := WORD#16#0015;   // $TC_MOP3[TOOL,3] CUTTING PREWARNING LIFE COUNTER
               BLOCKTYPE : Byte := BYTE#16#22;
               NUMOFLINE : Byte := BYTE#16#01;
               DATATYPE : Byte := BYTE#16#0F;
               LENGTH : Byte := BYTE#16#08;
            END_STRUCT;
            TC_MOP3_WARNING_4 : Struct
               SYNTAX_ID : Byte := BYTE#16#82;
               AREA_UNIT : Byte := BYTE#16#81;
               COLUMN : Word := 16#0;   // TOOL NUMBER (HEX)
               LINE : Word := WORD#16#001E;   // $TC_MOP3[TOOL,4] CUTTING PREWARNING LIFE COUNTER
               BLOCKTYPE : Byte := BYTE#16#22;
               NUMOFLINE : Byte := BYTE#16#01;
               DATATYPE : Byte := BYTE#16#0F;
               LENGTH : Byte := BYTE#16#08;
            END_STRUCT;
            TC_MOP3_WARNING_5 : Struct
               SYNTAX_ID : Byte := BYTE#16#82;
               AREA_UNIT : Byte := BYTE#16#81;
               COLUMN : Word := 16#0;   // TOOL NUMBER (HEX)
               LINE : Word := WORD#16#0027;   // $TC_MOP3[TOOL,4] CUTTING PREWARNING LIFE COUNTER / $TC_MOP3[TOOL,5] CUTTING PREWARNING LIFE COUNTER
               BLOCKTYPE : Byte := BYTE#16#22;
               NUMOFLINE : Byte := BYTE#16#01;
               DATATYPE : Byte := BYTE#16#0F;
               LENGTH : Byte := BYTE#16#08;
            END_STRUCT;
            TC_MOP13_EXPIRED_1 : Struct
               SYNTAX_ID : Byte := BYTE#16#82;
               AREA_UNIT : Byte := BYTE#16#81;
               COLUMN : Word := 16#0;   // TOOL NUMBER (HEX)
               LINE : Word := WORD#16#0006;   // $TC_MOP13[TOOL,1] CUTTING SET POINT LIFE COUNTER
               BLOCKTYPE : Byte := BYTE#16#22;
               NUMOFLINE : Byte := BYTE#16#01;
               DATATYPE : Byte := BYTE#16#0F;
               LENGTH : Byte := BYTE#16#08;
            END_STRUCT;
            TC_MOP13_EXPIRED_2 : Struct
               SYNTAX_ID : Byte := BYTE#16#82;
               AREA_UNIT : Byte := BYTE#16#81;
               COLUMN : Word := 16#0;   // TOOL NUMBER (HEX)
               LINE : Word := WORD#16#000F;   // $TC_MOP13[TOOL,2] CUTTING SET POINT LIFE COUNTER
               BLOCKTYPE : Byte := BYTE#16#22;
               NUMOFLINE : Byte := BYTE#16#01;
               DATATYPE : Byte := BYTE#16#0F;
               LENGTH : Byte := BYTE#16#08;
            END_STRUCT;
            TC_MOP13_EXPIRED_3 : Struct
               SYNTAX_ID : Byte := BYTE#16#82;
               AREA_UNIT : Byte := BYTE#16#81;
               COLUMN : Word := 16#0;   // TOOL NUMBER (HEX)
               LINE : Word := WORD#16#0018;   // $TC_MOP13[TOOL,3] CUTTING SET POINT LIFE COUNTER
               BLOCKTYPE : Byte := BYTE#16#22;
               NUMOFLINE : Byte := BYTE#16#01;
               DATATYPE : Byte := BYTE#16#0F;
               LENGTH : Byte := BYTE#16#08;
            END_STRUCT;
            TC_MOP13_EXPIRED_4 : Struct
               SYNTAX_ID : Byte := BYTE#16#82;
               AREA_UNIT : Byte := BYTE#16#81;
               COLUMN : Word := 16#0;   // TOOL NUMBER (HEX)
               LINE : Word := WORD#16#0021;   // $TC_MOP13[TOOL,4] CUTTING SET POINT LIFE COUNTER
               BLOCKTYPE : Byte := BYTE#16#22;
               NUMOFLINE : Byte := BYTE#16#01;
               DATATYPE : Byte := BYTE#16#0F;
               LENGTH : Byte := BYTE#16#08;
            END_STRUCT;
            TC_MOP13_EXPIRED_5 : Struct
               SYNTAX_ID : Byte := BYTE#16#82;
               AREA_UNIT : Byte := BYTE#16#81;
               COLUMN : Word := 16#0;   // TOOL NUMBER (HEX)
               LINE : Word := WORD#16#002A;   // $TC_MOP13[TOOL,4] CUTTING SET POINT LIFE COUNTER / $TC_MOP13[TOOL,5] CUTTING SET POINT LIFE COUNTER
               BLOCKTYPE : Byte := BYTE#16#22;
               NUMOFLINE : Byte := BYTE#16#01;
               DATATYPE : Byte := BYTE#16#0F;
               LENGTH : Byte := BYTE#16#08;
            END_STRUCT;
         END_STRUCT;
         PARAM_SPINDLE_SP2 : Struct
            TC_MOP4_QUANTITY_1 : Struct
               SYNTAX_ID : Byte := BYTE#16#82;
               AREA_UNIT : Byte := BYTE#16#81;
               COLUMN : Word := 16#0;   // TOOL NUMBER (HEX)
               LINE : Word := WORD#16#0004;   // $TC_MOP4[TOOL,1] CUTTING REMAINING LIFE COUNTER
               BLOCKTYPE : Byte := BYTE#16#22;
               NUMOFLINE : Byte := BYTE#16#01;
               DATATYPE : Byte := BYTE#16#0F;
               LENGTH : Byte := BYTE#16#08;
            END_STRUCT;
            TC_MOP4_QUANTITY_2 : Struct
               SYNTAX_ID : Byte := BYTE#16#82;
               AREA_UNIT : Byte := BYTE#16#81;
               COLUMN : Word := 16#0;   // TOOL NUMBER (HEX)
               LINE : Word := WORD#16#000D;   // $TC_MOP4[TOOL,2] CUTTING REMAINING LIFE COUNTER
               BLOCKTYPE : Byte := BYTE#16#22;
               NUMOFLINE : Byte := BYTE#16#01;
               DATATYPE : Byte := BYTE#16#0F;
               LENGTH : Byte := BYTE#16#08;
            END_STRUCT;
            TC_MOP4_QUANTITY_3 : Struct
               SYNTAX_ID : Byte := BYTE#16#82;
               AREA_UNIT : Byte := BYTE#16#81;
               COLUMN : Word := 16#0;   // TOOL NUMBER (HEX)
               LINE : Word := WORD#16#0016;   // $TC_MOP4[TOOL,3] CUTTING REMAINING LIFE COUNTER
               BLOCKTYPE : Byte := BYTE#16#22;
               NUMOFLINE : Byte := BYTE#16#01;
               DATATYPE : Byte := BYTE#16#0F;
               LENGTH : Byte := BYTE#16#08;
            END_STRUCT;
            TC_MOP4_QUANTITY_4 : Struct
               SYNTAX_ID : Byte := BYTE#16#82;
               AREA_UNIT : Byte := BYTE#16#81;
               COLUMN : Word := 16#0;   // TOOL NUMBER (HEX)
               LINE : Word := WORD#16#001F;   // $TC_MOP4[TOOL,4] CUTTING REMAINING LIFE COUNTER
               BLOCKTYPE : Byte := BYTE#16#22;
               NUMOFLINE : Byte := BYTE#16#01;
               DATATYPE : Byte := BYTE#16#0F;
               LENGTH : Byte := BYTE#16#08;
            END_STRUCT;
            TC_MOP4_QUANTITY_5 : Struct
               SYNTAX_ID : Byte := BYTE#16#82;
               AREA_UNIT : Byte := BYTE#16#81;
               COLUMN : Word := 16#0;   // TOOL NUMBER (HEX)
               LINE : Word := WORD#16#0028;   // $TC_MOP4[TOOL,4] CUTTING REMAINING LIFE COUNTER / $TC_MOP4[TOOL,5] CUTTING REMAINING LIFE COUNTER
               BLOCKTYPE : Byte := BYTE#16#22;
               NUMOFLINE : Byte := BYTE#16#01;
               DATATYPE : Byte := BYTE#16#0F;
               LENGTH : Byte := BYTE#16#08;
            END_STRUCT;
            TC_MOP3_WARNING_1 : Struct
               SYNTAX_ID : Byte := BYTE#16#82;
               AREA_UNIT : Byte := BYTE#16#81;
               COLUMN : Word := 16#0;   // TOOL NUMBER (HEX)
               LINE : Word := WORD#16#0003;   // $TC_MOP3[TOOL,1] CUTTING PREWARNING LIFE COUNTER
               BLOCKTYPE : Byte := BYTE#16#22;
               NUMOFLINE : Byte := BYTE#16#01;
               DATATYPE : Byte := BYTE#16#0F;
               LENGTH : Byte := BYTE#16#08;
            END_STRUCT;
            TC_MOP3_WARNING_2 : Struct
               SYNTAX_ID : Byte := BYTE#16#82;
               AREA_UNIT : Byte := BYTE#16#81;
               COLUMN : Word := 16#0;   // TOOL NUMBER (HEX)
               LINE : Word := WORD#16#000C;   // $TC_MOP3[TOOL,2] CUTTING PREWARNING LIFE COUNTER
               BLOCKTYPE : Byte := BYTE#16#22;
               NUMOFLINE : Byte := BYTE#16#01;
               DATATYPE : Byte := BYTE#16#0F;
               LENGTH : Byte := BYTE#16#08;
            END_STRUCT;
            TC_MOP3_WARNING_3 : Struct
               SYNTAX_ID : Byte := BYTE#16#82;
               AREA_UNIT : Byte := BYTE#16#81;
               COLUMN : Word := 16#0;   // TOOL NUMBER (HEX)
               LINE : Word := WORD#16#0015;   // $TC_MOP3[TOOL,3] CUTTING PREWARNING LIFE COUNTER
               BLOCKTYPE : Byte := BYTE#16#22;
               NUMOFLINE : Byte := BYTE#16#01;
               DATATYPE : Byte := BYTE#16#0F;
               LENGTH : Byte := BYTE#16#08;
            END_STRUCT;
            TC_MOP3_WARNING_4 : Struct
               SYNTAX_ID : Byte := BYTE#16#82;
               AREA_UNIT : Byte := BYTE#16#81;
               COLUMN : Word := 16#0;   // TOOL NUMBER (HEX)
               LINE : Word := WORD#16#001E;   // $TC_MOP3[TOOL,4] CUTTING PREWARNING LIFE COUNTER
               BLOCKTYPE : Byte := BYTE#16#22;
               NUMOFLINE : Byte := BYTE#16#01;
               DATATYPE : Byte := BYTE#16#0F;
               LENGTH : Byte := BYTE#16#08;
            END_STRUCT;
            TC_MOP3_WARNING_5 : Struct
               SYNTAX_ID : Byte := BYTE#16#82;
               AREA_UNIT : Byte := BYTE#16#81;
               COLUMN : Word := 16#0;   // TOOL NUMBER (HEX)
               LINE : Word := WORD#16#0027;   // $TC_MOP3[TOOL,4] CUTTING PREWARNING LIFE COUNTER / $TC_MOP3[TOOL,5] CUTTING PREWARNING LIFE COUNTER
               BLOCKTYPE : Byte := BYTE#16#22;
               NUMOFLINE : Byte := BYTE#16#01;
               DATATYPE : Byte := BYTE#16#0F;
               LENGTH : Byte := BYTE#16#08;
            END_STRUCT;
            TC_MOP13_EXPIRED_1 : Struct
               SYNTAX_ID : Byte := BYTE#16#82;
               AREA_UNIT : Byte := BYTE#16#81;
               COLUMN : Word := 16#0;   // TOOL NUMBER (HEX)
               LINE : Word := WORD#16#0006;   // $TC_MOP13[TOOL,1] CUTTING SET POINT LIFE COUNTER
               BLOCKTYPE : Byte := BYTE#16#22;
               NUMOFLINE : Byte := BYTE#16#01;
               DATATYPE : Byte := BYTE#16#0F;
               LENGTH : Byte := BYTE#16#08;
            END_STRUCT;
            TC_MOP13_EXPIRED_2 : Struct
               SYNTAX_ID : Byte := BYTE#16#82;
               AREA_UNIT : Byte := BYTE#16#81;
               COLUMN : Word := 16#0;   // TOOL NUMBER (HEX)
               LINE : Word := WORD#16#000F;   // $TC_MOP13[TOOL,2] CUTTING SET POINT LIFE COUNTER
               BLOCKTYPE : Byte := BYTE#16#22;
               NUMOFLINE : Byte := BYTE#16#01;
               DATATYPE : Byte := BYTE#16#0F;
               LENGTH : Byte := BYTE#16#08;
            END_STRUCT;
            TC_MOP13_EXPIRED_3 : Struct
               SYNTAX_ID : Byte := BYTE#16#82;
               AREA_UNIT : Byte := BYTE#16#81;
               COLUMN : Word := 16#0;   // TOOL NUMBER (HEX)
               LINE : Word := WORD#16#0018;   // $TC_MOP13[TOOL,3] CUTTING SET POINT LIFE COUNTER
               BLOCKTYPE : Byte := BYTE#16#22;
               NUMOFLINE : Byte := BYTE#16#01;
               DATATYPE : Byte := BYTE#16#0F;
               LENGTH : Byte := BYTE#16#08;
            END_STRUCT;
            TC_MOP13_EXPIRED_4 : Struct
               SYNTAX_ID : Byte := BYTE#16#82;
               AREA_UNIT : Byte := BYTE#16#81;
               COLUMN : Word := 16#0;   // TOOL NUMBER (HEX)
               LINE : Word := WORD#16#0021;   // $TC_MOP13[TOOL,4] CUTTING SET POINT LIFE COUNTER
               BLOCKTYPE : Byte := BYTE#16#22;
               NUMOFLINE : Byte := BYTE#16#01;
               DATATYPE : Byte := BYTE#16#0F;
               LENGTH : Byte := BYTE#16#08;
            END_STRUCT;
            TC_MOP13_EXPIRED_5 : Struct
               SYNTAX_ID : Byte := BYTE#16#82;
               AREA_UNIT : Byte := BYTE#16#81;
               COLUMN : Word := 16#0;   // TOOL NUMBER (HEX)
               LINE : Word := WORD#16#002A;   // $TC_MOP13[TOOL,4] CUTTING SET POINT LIFE COUNTER / $TC_MOP13[TOOL,5] CUTTING SET POINT LIFE COUNTER
               BLOCKTYPE : Byte := BYTE#16#22;
               NUMOFLINE : Byte := BYTE#16#01;
               DATATYPE : Byte := BYTE#16#0F;
               LENGTH : Byte := BYTE#16#08;
            END_STRUCT;
         END_STRUCT;
         FB2_VARS_SP1 : Struct
            TOOL_NUMBER : Struct
               error : Bool;
               done : Bool;
               request : Bool;
            END_STRUCT;
            ORIGI_MAGAZINE : Struct
               error : Bool;
               done : Bool;
               request : Bool;
            END_STRUCT;
            CUTING_EDGE : Struct
               error : Bool;
               done : Bool;
               request : Bool;
            END_STRUCT;
            QUANTITY_EDGE : Struct
               error : Bool;
               done : Bool;
               request : Bool;
            END_STRUCT;
            WARNING_EDGE : Struct
               error : Bool;
               done : Bool;
               request : Bool;
            END_STRUCT;
            EXPIRED_EDGE : Struct
               error : Bool;
               done : Bool;
               request : Bool;
            END_STRUCT;
         END_STRUCT;
         FB2_VARS_SP2 : Struct
            TOOL_NUMBER : Struct
               error : Bool;
               done : Bool;
               request : Bool;
            END_STRUCT;
            ORIGI_MAGAZINE : Struct
               error : Bool;
               done : Bool;
               request : Bool;
            END_STRUCT;
            CUTING_EDGE : Struct
               error : Bool;
               done : Bool;
               request : Bool;
            END_STRUCT;
            QUANTITY_EDGE : Struct
               error : Bool;
               done : Bool;
               request : Bool;
            END_STRUCT;
            WARNING_EDGE : Struct
               error : Bool;
               done : Bool;
               request : Bool;
            END_STRUCT;
            EXPIRED_EDGE : Struct
               error : Bool;
               done : Bool;
               request : Bool;
            END_STRUCT;
         END_STRUCT;
         SMNS_PRMTRS_SP1 : Struct
            TC_MPP6_PLACE_DATA : Struct
               SYNTAX_ID : Byte := BYTE#16#82;
               AREA_UNIT : Byte := BYTE#16#81;   // CHANNEL NUMBER, 81=CH1, 82=CH2 )
               COLUMN : Word := WORD#16#0001;   // MAGAZINE NUMBER
               LINE : Word := 16#0;
               BLOCKTYPE : Byte := BYTE#16#28;
               NUMOFLINE : Byte := BYTE#16#01;
               DATATYPE : Byte := BYTE#16#04;
               LENGTH : Byte := BYTE#16#02;
            END_STRUCT;
            NUM_CUTTING_EDGES : Struct
               SYNTAX_ID : Byte := BYTE#16#82;
               AREA_UNIT : Byte := BYTE#16#81;
               COLUMN : Word := WORD#16#000E;   // NUM CUTTING EDGES
               LINE : Word := WORD#16#0001;
               BLOCKTYPE : Byte := BYTE#16#21;
               NUMOFLINE : Byte := BYTE#16#01;
               DATATYPE : Byte := BYTE#16#04;
               LENGTH : Byte := BYTE#16#02;
            END_STRUCT;
            DUPLO_NUMBER : Struct
               SYNTAX_ID : Byte := BYTE#16#82;
               AREA_UNIT : Byte := BYTE#16#81;
               COLUMN : Word := WORD#16#0002;   // DUPLO NUMBER
               LINE : Word := WORD#16#0001;
               BLOCKTYPE : Byte := BYTE#16#21;
               NUMOFLINE : Byte := BYTE#16#01;
               DATATYPE : Byte := BYTE#16#04;
               LENGTH : Byte := BYTE#16#02;
            END_STRUCT;
            ORIG_MAGAZINE : Struct
               SYNTAX_ID : Byte := BYTE#16#82;
               AREA_UNIT : Byte := BYTE#16#81;
               COLUMN : Word := WORD#16#0011;   // ORIG MAGAZINE
               LINE : Word := WORD#16#0001;
               BLOCKTYPE : Byte := BYTE#16#21;
               NUMOFLINE : Byte := BYTE#16#01;
               DATATYPE : Byte := BYTE#16#04;
               LENGTH : Byte := BYTE#16#02;
            END_STRUCT;
         END_STRUCT;
         SMNS_PRMTRS_SP2 : Struct
            TC_MPP6_PLACE_DATA : Struct
               SYNTAX_ID : Byte := BYTE#16#82;
               AREA_UNIT : Byte := BYTE#16#81;   // CHANNEL NUMBER, 81=CH1, 82=CH2 )
               COLUMN : Word := WORD#16#0001;   // MAGAZINE NUMBER
               LINE : Word := 16#0;
               BLOCKTYPE : Byte := BYTE#16#28;
               NUMOFLINE : Byte := BYTE#16#01;
               DATATYPE : Byte := BYTE#16#04;
               LENGTH : Byte := BYTE#16#02;
            END_STRUCT;
            NUM_CUTTING_EDGES : Struct
               SYNTAX_ID : Byte := BYTE#16#82;
               AREA_UNIT : Byte := BYTE#16#81;
               COLUMN : Word := WORD#16#000E;   // NUM CUTTING EDGES
               LINE : Word := WORD#16#0001;
               BLOCKTYPE : Byte := BYTE#16#21;
               NUMOFLINE : Byte := BYTE#16#01;
               DATATYPE : Byte := BYTE#16#04;
               LENGTH : Byte := BYTE#16#02;
            END_STRUCT;
            DUPLO_NUMBER : Struct
               SYNTAX_ID : Byte := BYTE#16#82;
               AREA_UNIT : Byte := BYTE#16#81;
               COLUMN : Word := WORD#16#0002;   // DUPLO NUMBER
               LINE : Word := WORD#16#0001;
               BLOCKTYPE : Byte := BYTE#16#21;
               NUMOFLINE : Byte := BYTE#16#01;
               DATATYPE : Byte := BYTE#16#04;
               LENGTH : Byte := BYTE#16#02;
            END_STRUCT;
            ORIG_MAGAZINE : Struct
               SYNTAX_ID : Byte := BYTE#16#82;
               AREA_UNIT : Byte := BYTE#16#81;
               COLUMN : Word := WORD#16#0011;   // ORIG MAGAZINE
               LINE : Word := WORD#16#0001;
               BLOCKTYPE : Byte := BYTE#16#21;
               NUMOFLINE : Byte := BYTE#16#01;
               DATATYPE : Byte := BYTE#16#04;
               LENGTH : Byte := BYTE#16#02;
            END_STRUCT;
         END_STRUCT;
      END_STRUCT;
   END_STRUCT;
   // // READ.TOOL_DATA_SP1.QUANTITY_EDGE[1] : QUANTITY EDGE[1]
   // // READ.TOOL_DATA_SP1.QUANTITY_EDGE[2] : QUANTITY EDGE[2]
   // // READ.TOOL_DATA_SP1.QUANTITY_EDGE[3] : QUANTITY EDGE[3]
   // // READ.TOOL_DATA_SP1.QUANTITY_EDGE[4] : QUANTITY EDGE[4]
   // // READ.TOOL_DATA_SP1.QUANTITY_EDGE[5] : QUANTITY EDGE[5]
   // // READ.TOOL_DATA_SP1.WARNING_EDGE[1] : WARNING EDGE[1]
   // // READ.TOOL_DATA_SP1.WARNING_EDGE[2] : WARNING EDGE[2]
   // // READ.TOOL_DATA_SP1.WARNING_EDGE[3] : WARNING EDGE[3]
   // // READ.TOOL_DATA_SP1.WARNING_EDGE[4] : WARNING EDGE[4]
   // // READ.TOOL_DATA_SP1.WARNING_EDGE[5] : WARNING EDGE[5]
   // // READ.TOOL_DATA_SP1.EXPIRED_EDGE[1] : EXPIRED EDGE[1]
   // // READ.TOOL_DATA_SP1.EXPIRED_EDGE[2] : EXPIRED EDGE[2]
   // // READ.TOOL_DATA_SP1.EXPIRED_EDGE[3] : EXPIRED EDGE[3]
   // // READ.TOOL_DATA_SP1.EXPIRED_EDGE[4] : EXPIRED EDGE[4]
   // // READ.TOOL_DATA_SP1.EXPIRED_EDGE[5] : EXPIRED EDGE[5]
   // // READ.TOOL_DATA_SP2.QUANTITY_EDGE[1] : QUANTITY EDGE[1]
   // // READ.TOOL_DATA_SP2.QUANTITY_EDGE[2] : QUANTITY EDGE[2]
   // // READ.TOOL_DATA_SP2.QUANTITY_EDGE[3] : QUANTITY EDGE[3]
   // // READ.TOOL_DATA_SP2.QUANTITY_EDGE[4] : QUANTITY EDGE[4]
   // // READ.TOOL_DATA_SP2.QUANTITY_EDGE[5] : QUANTITY EDGE[5]
   // // READ.TOOL_DATA_SP2.WARNING_EDGE[1] : WARNING EDGE[1]
   // // READ.TOOL_DATA_SP2.WARNING_EDGE[2] : WARNING EDGE[2]
   // // READ.TOOL_DATA_SP2.WARNING_EDGE[3] : WARNING EDGE[3]
   // // READ.TOOL_DATA_SP2.WARNING_EDGE[4] : WARNING EDGE[4]
   // // READ.TOOL_DATA_SP2.WARNING_EDGE[5] : WARNING EDGE[5]
   // // READ.TOOL_DATA_SP2.EXPIRED_EDGE[1] : EXPIRED EDGE[1]
   // // READ.TOOL_DATA_SP2.EXPIRED_EDGE[2] : EXPIRED EDGE[2]
   // // READ.TOOL_DATA_SP2.EXPIRED_EDGE[3] : EXPIRED EDGE[3]
   // // READ.TOOL_DATA_SP2.EXPIRED_EDGE[4] : EXPIRED EDGE[4]
   // // READ.TOOL_DATA_SP2.EXPIRED_EDGE[5] : EXPIRED EDGE[5]
END_TYPE

